GLOBALCONSTANTS AID_OS (* Output string object attribute ids *)
  (* Standard: 61499-1; Description: Copyright (c) 2023 HR Agrartechnik GmbH This program and the accompanying materials are made available under the terms of the Eclipse Public License 2.0 which is available at https://www.eclipse.org/legal/epl-2.0/ SPDX-License-Identifier: EPL-2.0 *)
  (* Version 1.0, 2026-06-20, Franz Höpfinger, HR Agrartechnik GmbH *)
  PACKAGE isobus::UT::Q::const::AID;
  IMPORT eclipse4diac::core::TypeHash;
  VAR_GLOBAL CONSTANT
    WIDTH : USINT := USINT#1; (* 1: AID_OS_WIDTH - Width in pixels. *)
    HEIGHT : USINT := USINT#2; (* 2: AID_OS_HEIGHT - Height in pixels. *)
    BACKGROUND_COLOUR : USINT := USINT#3; (* 3: AID_OS_BACKGROUND_COLOUR - Background colour index. *)
    FONT_ATT : USINT := USINT#4; (* 4: AID_OS_FONT_ATT - Object ID of a Font Attributes object. *)
    OPTIONS : USINT := USINT#5; (* 5: AID_OS_OPTIONS - Bitmask: Bit 0=Transparent, Bit 1=Auto-Wrap, Bit 2=Wrap on Hyphen. *)
    VARIABLE_REF : USINT := USINT#6; (* 6: AID_OS_VARIABLE_REF - Object ID of a Variable object. *)
    JUSTIFICATION : USINT := USINT#7; (* 7: AID_OS_JUSTIFICATION - Justification: Bits 0-1 (Horizontal: 0=Left, 1=Middle, 2=Right), Bits 2-3 (Vertical: 0=Top, 1=Middle, 2=Bottom). *)
  END_VAR
END_GLOBALCONSTANTS
